Fanuc TP program (LS listing): LASON.LS

/PROG  LASON
/ATTR
OWNER		= MNEDITOR;
COMMENT		= "";
PROG_SIZE	= 167;
CREATE		= DATE 80-01-01  TIME 00:37:20;
MODIFIED	= DATE 80-01-01  TIME 00:37:50;
FILE_NAME	= ;
VERSION		= 0;
LINE_COUNT	= 1;
MEMORY_SIZE	= 535;
PROTECT		= READ_WRITE;
TCD:  STACK_SIZE	= 0,
      TASK_PRIORITY	= 50,
      TIME_SLICE	= 0,
      BUSY_LAMP_OFF	= 0,
      ABORT_REQUEST	= 0,
      PAUSE_REQUEST	= 0;
DEFAULT_GROUP	= 1,*,*,*,*;
CONTROL_CODE	= 00000000 00000000;
/APPL
  ARC Welding Equipment : 1,*,*,*,*;
/MN
   1:  SENSOR ON[1] ;
/POS
/END
